(* PLC project SafeLOGIC-1, BrAutomation SafeDESIGNER  4.4.0.0 *)
(* stored: companyURL http://www.br-automation.com, creationDateTime Fri Aug 20 07:50:25 2021 *)

PROGRAM Main

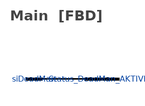
(* FBD diagram, written out as Structured Text *)
Status_DeadMan_AKTIVNY := siDeadMan;
END_PROGRAM
